Universal Robots PolyScope program: Arla0.4.urp

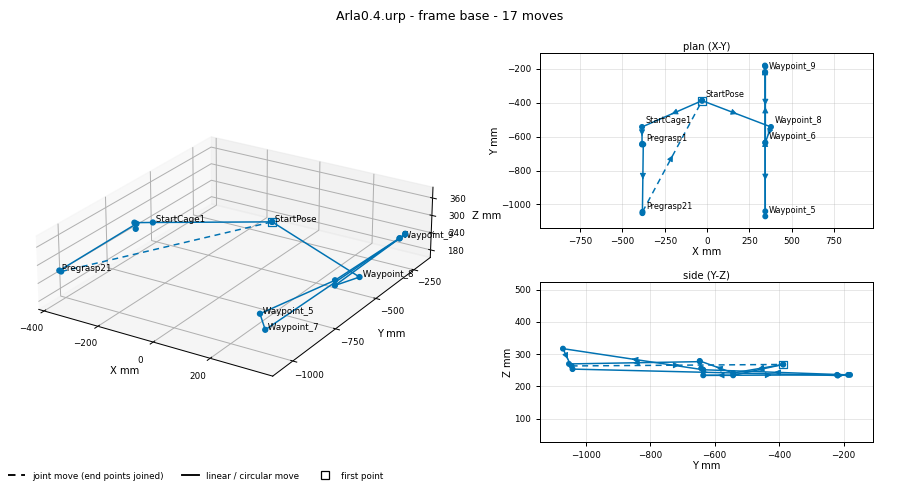
[picture p0: tool path of Arla0.4.urp in frame base, 17 of 17 moves have a stored position in this frame; points joined in program order, loops and branches not executed]
Program Arla0.4 (installation=default directory=/programs/usbdisk_0 createdIn=5.11.4.108353 lastSavedIn=5.9.1.1031110 robotSerialNumber=20185000125)
Calibrated DH parameters: a=[0.000009, -0.582937, -0.560313, -0.000136, -0.000015, 0]; d=[0.181003, 62.966139, -25.546705, -37.245036, 0.119984, 0.115761]; alpha=[1.570753, -0.002987, -0.002977, 1.572291, -1.570292, 0]; deltaTheta=[-0.000001, -0.312112, 0.115839, 0.196276, -0.000002, 0]
Robot Program (runOnlyOnce=true)
  Folder ResetForce
    Wait Condition expression=is_steady()
    Wait Sleep waitTime=0.25
    Script: zero_ftsensor()
    Wait Sleep waitTime=0.25
  Timer (action=Start) variable(name=timer_1)
  MoveJ speed 30 deg/s, acceleration 40 deg/s^2 (useActiveTCP=true) feature=Base
    Waypoint StartPose: motionParameters(jointSpeed=0.523599 jointAcceleration=0.698132 cartesianSpeed=0.25 cartesianAcceleration=1.2); TCP in base x=-29.649 y=-387.378 z=267.725 mm, rx=0 ry=-3.1416 rz=0 rad; joints [-67.884, -70.586, -150.404, -49.041, 89.902, 22.237] deg
  Folder Cage1
    MoveL speed 250 mm/s, acceleration 1200 mm/s^2 (useActiveTCP=true) feature=Base
      Waypoint StartCage1: TCP in base x=-384.45 y=-542.641 z=241.291 mm, rx=-0.1647 ry=-3.1372 rz=0.0005 rad; joints [-110.238, -102.782, -124.633, -42.597, 89.826, -14.14] deg
    MoveL speed 250 mm/s, acceleration 1200 mm/s^2 (useActiveTCP=true) feature=Base
      Waypoint Pregrasp1: TCP in base x=-384.451 y=-646.287 z=278.645 mm, rx=-0.1639 ry=-3.1201 rz=-0.2382 rad; joints [-107.053, -107.186, -111.215, -59.984, 87.241, -10.726] deg
    MoveL speed 250 mm/s, acceleration 1200 mm/s^2 (useActiveTCP=true) feature=Base
      Waypoint Waypoint_1: TCP in base x=-383.037 y=-641.745 z=255.803 mm, rx=-0.1626 ry=-3.1373 rz=-0.0001 rad; joints [-107.451, -108.111, -115.055, -46.865, 89.802, -11.433] deg
    Set DigitalOutput pin=digital_out[0]; digitalValue=1
    Wait Sleep waitTime=0.7
    var_1 := get_actual_tcp_pose()
    Force Frame feature=Base; selection=[0, 0, 1, 0, 0, 0]; wrench=[0, 10, 225, 0, 0, 0]; limitsForce=[0.15, 0.15, 0.15, 1.047198, 1.047198, 1.047198]; limitsMotion=[0.1, 0.1, 0.1, 0.349066, 0.349066, 0.349066]
      Loop While (checkContinuously=false) expression=var_1[2] < 0.275
        var_1 := get_actual_tcp_pose()
    MoveL speed 100 mm/s, acceleration 1200 mm/s^2 (useActiveTCP=true) feature=Base
      MoveDirectionNode (selectedDirection=YPlus)
        Until DISTANCE (allowActions=false deceleration=3 distanceNodeType=STOP) Distance=0.1; motionParameters(blendRadius=0)
    Set DigitalOutput pin=digital_out[0]; digitalValue=0
    MoveL speed 100 mm/s, acceleration 1200 mm/s^2 (useActiveTCP=true) feature=Base
      MoveDirectionNode (selectedDirection=YPlus)
        Until DISTANCE (allowActions=false deceleration=3 distanceNodeType=STOP) Distance=0.17; motionParameters(blendRadius=0)
    MoveL speed 200 mm/s, acceleration 400 mm/s^2 (useActiveTCP=true) feature=Base
      MoveDirectionNode (selectedDirection=ZMinus)
        Until DISTANCE (allowActions=false deceleration=3 distanceNodeType=STOP) Distance=0.012; motionParameters(blendRadius=0)
    MoveL speed 200 mm/s, acceleration 400 mm/s^2 (useActiveTCP=true) feature=Base
      MoveDirectionNode (selectedDirection=YPlus)
        Until DISTANCE (allowActions=false deceleration=3 distanceNodeType=STOP) Distance=0.165; motionParameters(blendRadius=0)
    MoveL speed 200 mm/s, acceleration 400 mm/s^2 (useActiveTCP=true) feature=Base
      MoveDirectionNode (selectedDirection=ZMinus)
        Until DISTANCE (allowActions=false deceleration=3 distanceNodeType=STOP) Distance=0.025; motionParameters(blendRadius=0)
    MoveL speed 200 mm/s, acceleration 400 mm/s^2 (useActiveTCP=true) feature=Base
      MoveDirectionNode (selectedDirection=YPlus)
        Until DISTANCE (allowActions=false deceleration=3 distanceNodeType=STOP) Distance=0.05; motionParameters(blendRadius=0)
    Halt
    MoveL speed 250 mm/s, acceleration 1200 mm/s^2 (useActiveTCP=true) feature=Base
      Waypoint Waypoint_14: TCP in base x=-377.026 y=-645.668 z=276.467 mm, rx=0.1472 ry=3.1381 rz=-0.0003 rad; joints [-106.91, -106.71, -114.273, -49.036, 89.805, -11.447] deg
    MoveL speed 250 mm/s, acceleration 1200 mm/s^2 (useActiveTCP=true) feature=Base
      Waypoint Pregrasp21: TCP in base x=-382.3 y=-1051.922 z=269.368 mm, rx=-0.1465 ry=-3.1225 rz=-0.2333 rad; joints [-100.889, -138.911, -59.571, -79.947, 88.091, -5.286] deg
    MoveL speed 300 mm/s, acceleration 1200 mm/s^2 (useActiveTCP=true) feature=Base
      Waypoint Pregrasp22: TCP in base x=-381.59 y=-1043.818 z=263.117 mm, rx=0.1466 ry=3.1279 rz=0.0097 rad; joints [-101.159, -137.268, -64.922, -68.277, 90.233, -5.728] deg
    MoveL speed 250 mm/s, acceleration 1200 mm/s^2 (useActiveTCP=true) feature=Base
      MoveDirectionNode (selectedDirection=YPlus)
        Until DISTANCE (allowActions=false deceleration=3 distanceNodeType=STOP) Distance=0.405; motionParameters(blendRadius=0)
    var_1 := get_actual_tcp_pose()
    Force Frame feature=Base; selection=[0, 0, 1, 0, 0, 0]; wrench=[0, 10, 225, 0, 0, 0]; limitsForce=[0.15, 0.15, 0.15, 1.047198, 1.047198, 1.047198]; limitsMotion=[0.1, 0.1, 0.1, 0.349066, 0.349066, 0.349066]
      Loop While (checkContinuously=false) expression=var_1[2] < 0.278
        var_1 := get_actual_tcp_pose()
    MoveL speed 200 mm/s, acceleration 400 mm/s^2 (useActiveTCP=true) feature=Base
      MoveDirectionNode (selectedDirection=YPlus)
        Until DISTANCE (allowActions=false deceleration=3 distanceNodeType=STOP) Distance=0.25; motionParameters(blendRadius=0)
    MoveL speed 100 mm/s, acceleration 400 mm/s^2 (useActiveTCP=true) feature=Base
      MoveDirectionNode (selectedDirection=ZMinus)
        Until DISTANCE (allowActions=false deceleration=3 distanceNodeType=STOP) Distance=0.015; motionParameters(blendRadius=0)
    Wait Sleep waitTime=0.5
    MoveL speed 200 mm/s, acceleration 400 mm/s^2 (useActiveTCP=true) feature=Base
      MoveDirectionNode (selectedDirection=YPlus)
        Until DISTANCE (allowActions=false deceleration=3 distanceNodeType=STOP) Distance=0.185; motionParameters(blendRadius=0)
    MoveL speed 200 mm/s, acceleration 400 mm/s^2 (useActiveTCP=true) feature=Base
      MoveDirectionNode (selectedDirection=ZMinus)
        Until DISTANCE (allowActions=false deceleration=3 distanceNodeType=STOP) Distance=0.025; motionParameters(blendRadius=0)
    MoveL speed 200 mm/s, acceleration 400 mm/s^2 (useActiveTCP=true) feature=Base
      MoveDirectionNode (selectedDirection=YPlus)
        Until DISTANCE (allowActions=false deceleration=3 distanceNodeType=STOP) Distance=0.05; motionParameters(blendRadius=0)
    Halt
    Wait Sleep waitTime=2
  MoveJ speed 30 deg/s, acceleration 40 deg/s^2 (useActiveTCP=true) feature=Base
    Waypoint StartPose: motionParameters(jointSpeed=0.523599 jointAcceleration=0.698132 cartesianSpeed=0.25 cartesianAcceleration=1.2); TCP in base x=-29.649 y=-387.378 z=267.725 mm, rx=0 ry=-3.1416 rz=0 rad; joints [-67.884, -70.586, -150.404, -49.041, 89.902, 22.237] deg
  Timer (action=Start) variable=timer_1
  Halt
  Folder Cage2
    MoveL speed 400 mm/s, acceleration 1200 mm/s^2 (useActiveTCP=true) feature=Base
      Waypoint Waypoint_8: TCP in base x=377.02 y=-542.594 z=233.918 mm, rx=-0.1647 ry=-3.1372 rz=0.0003 rad; joints [-40.025, -103.065, -125.347, -41.613, 89.819, 56.073] deg; TCP offset x=0 y=0 z=0 mm, rx=0 ry=0 rz=0 rad
    MoveL speed 400 mm/s, acceleration 1200 mm/s^2 (useActiveTCP=true) feature=Base
      Waypoint Waypoint_6: TCP in base x=343.499 y=-635.479 z=233.957 mm, rx=-0.1647 ry=-3.1373 rz=0.0004 rad; joints [-47.751, -107.813, -118.586, -43.62, 89.801, 48.338] deg
    Set DigitalOutput pin=digital_out[0]; digitalValue=1
    var_1 := get_actual_tcp_pose()
    Force Frame feature=Base; selection=[0, 0, 1, 0, 0, 0]; wrench=[0, 10, 225, 0, 0, 0]; limitsForce=[0.15, 0.15, 0.15, 1.047198, 1.047198, 1.047198]; limitsMotion=[0.1, 0.1, 0.1, 0.349066, 0.349066, 0.349066]
      Loop While (checkContinuously=false) expression=var_1[2] < 0.275
        var_1 := get_actual_tcp_pose()
    var_1 := get_actual_tcp_pose()
    Force Frame feature=Base; selection=[0, 0, 1, 0, 0, 0]; wrench=[0, 10, 225, 0, 0, 0]; limitsForce=[0.15, 0.15, 0.15, 1.047198, 1.047198, 1.047198]; limitsMotion=[0.1, 0.1, 0.1, 0.349066, 0.349066, 0.349066]
      Set DigitalOutput pin=digital_out[0]; digitalValue=1
    MoveL speed 250 mm/s, acceleration 1200 mm/s^2 (useActiveTCP=true) feature=Base
      MoveDirectionNode (selectedDirection=YPlus)
        Until DISTANCE (allowActions=false deceleration=3 distanceNodeType=STOP) Distance=0.1; motionParameters(blendRadius=0)
    Set DigitalOutput pin=digital_out[0]; digitalValue=0
    MoveL speed 200 mm/s, acceleration 1200 mm/s^2 (useActiveTCP=true) feature=Base
      MoveDirectionNode (selectedDirection=YPlus)
        Until DISTANCE (allowActions=false deceleration=3 distanceNodeType=STOP) Distance=0.315; motionParameters(blendRadius=0)
    MoveL speed 400 mm/s, acceleration 1200 mm/s^2 (useActiveTCP=true) feature=Base
      Waypoint Waypoint_9: TCP in base x=343.344 y=-220.193 z=235.398 mm, rx=-0.1642 ry=-3.1366 rz=-0.0011 rad; joints [-7.535, -77.835, -150.69, -41.549, 89.937, 88.568] deg
    MoveL speed 400 mm/s, acceleration 1200 mm/s^2 (useActiveTCP=true) feature=Base
      Waypoint Waypoint_10: TCP in base x=343.967 y=-185.915 z=235.406 mm, rx=-0.1641 ry=-3.1366 rz=-0.0011 rad; joints [-2.083, -75.381, -152.234, -42.453, 89.944, 94.019] deg
    MoveL speed 400 mm/s, acceleration 1200 mm/s^2 (useActiveTCP=true) feature=Base
      Waypoint Waypoint_11: TCP in base x=343.517 y=-635.445 z=251.337 mm, rx=-0.1646 ry=-3.1372 rz=0.0002 rad; joints [-47.75, -106.495, -118.012, -45.518, 89.802, 48.342] deg
    MoveL speed 400 mm/s, acceleration 1200 mm/s^2 (useActiveTCP=true) feature=Base
      Waypoint Waypoint_5: TCP in base x=343.517 y=-1070.669 z=316.765 mm, rx=-0.1606 ry=-3.064 rz=-0.5775 rad; joints [-64.275, -141.022, -49.138, -99.241, 98.786, 30.359] deg
    MoveL speed 400 mm/s, acceleration 1200 mm/s^2 (useActiveTCP=true) feature=Base
      Waypoint Waypoint_7: TCP in base x=343.552 y=-1041.014 z=253.298 mm, rx=-0.1644 ry=-3.1372 rz=0.0001 rad; joints [-62.635, -136.166, -68.133, -65.731, 89.702, 33.426] deg
    MoveL speed 400 mm/s, acceleration 1200 mm/s^2 (useActiveTCP=true) feature=Base
      MoveDirectionNode (selectedDirection=YPlus)
        Until DISTANCE (allowActions=false deceleration=3 distanceNodeType=STOP) Distance=0.405; motionParameters(blendRadius=0)
    var_1 := get_actual_tcp_pose()
    Force Frame feature=Base; selection=[0, 0, 1, 0, 0, 0]; wrench=[0, 10, 225, 0, 0, 0]; limitsForce=[0.15, 0.15, 0.15, 1.047198, 1.047198, 1.047198]; limitsMotion=[0.1, 0.1, 0.1, 0.349066, 0.349066, 0.349066]
      Loop While (checkContinuously=false) expression=var_1[2] < 0.275
        var_1 := get_actual_tcp_pose()
    Wait Sleep waitTime=0.5
    MoveL speed 200 mm/s, acceleration 400 mm/s^2 (useActiveTCP=true) feature=Base
      MoveDirectionNode (selectedDirection=YPlus)
        Until DISTANCE (allowActions=false deceleration=3 distanceNodeType=STOP) Distance=0.415; motionParameters(blendRadius=0.05)
    MoveL speed 400 mm/s, acceleration 1200 mm/s^2 (useActiveTCP=true) feature=Base
      Waypoint Waypoint_12: TCP in base x=341.332 y=-218.663 z=233.476 mm, rx=-0.1641 ry=-3.132 rz=-0.007 rad; joints [-7.4, -77.77, -150.937, -41.641, 90.132, 88.707] deg
    MoveL speed 400 mm/s, acceleration 1200 mm/s^2 (useActiveTCP=true) feature=Base
      Waypoint Waypoint_13: TCP in base x=341.336 y=-179.93 z=235.41 mm, rx=-0.164 ry=-3.132 rz=-0.007 rad; joints [-1.184, -74.618, -152.606, -43.097, 90.172, 94.922] deg
  Timer (action=Stop) variable=timer_1
